(* concatenate 3 strings *)
FUNCTION F_CONCAT3 : T_MaxString
VAR_INPUT
	strString1		: T_MaxString;
	strString2		: T_MaxString;
	strString3		: T_MaxString;
END_VAR
VAR
END_VAR
(*
-------------------------------------------------------------------------------------------------
Date		Version	Author	Comments
-------------------------------------------------------------------------------------------------
30/01/2015	3.00.00	PB		No change

-------------------------------------------------------------------------------------------------
05/02/2010	1.00.00	PB		Initial release

-------------------------------------------------------------------------------------------------
*)

F_CONCAT3 := CONCAT(strString1, strString2);
F_CONCAT3 := CONCAT(F_CONCAT3, strString3);

END_FUNCTION

(* stored: Version 1.1.0.1, ProductVersion 3.1.4024.15
   POU F_CONCAT3: Id {e9dce370-253d-421c-97c8-7de3d83ece43}, SpecialFunc None *)
